FUNCTION_BLOCK ConveyorSC_NC
VAR_INPUT
	bEnable : BOOL;
END_VAR
VAR_OUTPUT
	sensorEntry AT %I* : BOOL := TRUE;
	sensorExit AT %I* : BOOL := TRUE;
	
	trueMode : ConveyorMode;
	requestedMode : ConveyorMode;
	
	position : LREAL;
	velocity : LREAL;
	ready : BOOL;
END_VAR
VAR
	axis : AXIS_REF;
	
	mcReadPosition : MC_ReadActualPosition; //continuous enable FBs
	mcReadVelocity : MC_ReadActualVelocity;
	mcReadError : MC_ReadAxisError;
	mcPower : MC_Power;
	
	mcReset : MC_Reset; //rising edge FBs
	mcMoveAbsolute : MC_MoveAbsolute;
	mcMoveRelative : MC_MoveRelative;
	mcMoveVelocity : MC_MoveVelocity;
	
	mcSetPosition : MC_SetPosition;
	mcStop : MC_Stop;
END_VAR
VAR_STAT CONSTANT
	targetingVelocity : INT := 500;
	continuousVelocity : INT := 500;
END_VAR
(*
this FB represents a standard slat conveyor with no lifter
	compliant with PLCopen motion control

unlike standalone servos,
	conveyors need to coordinate (not slave) their motion with other conveyors
	and be able to set their current position to any value as required by the system
	
moveAbsolute is provided for now but should not be used for position targetting and may be protected/privated later
instead, request/set the operation mode and the motion will follow
*)

IF error THEN
	stop();
	reset();
	
ELSE
	CASE trueMode OF
		ConveyorMode.IDLE:			stop();	
		ConveyorMode.FORWARD:		moveContinuous(direction:= MC_Positive_Direction);
		ConveyorMode.BACKWARD:		moveContinuous(direction:= MC_Negative_Direction);
		ConveyorMode.STOP:			stop();
	END_CASE
	
END_IF

blocks();

mcReset.Execute := FALSE;
mcMoveAbsolute.Execute := FALSE;
mcMoveRelative.Execute := FALSE;
mcMoveVelocity.Execute := FALSE;
mcSetPosition.Execute := FALSE;
mcStop.Execute := FALSE;

blocks();

PROPERTY Active : BOOL
GET
Active := 
	mcMoveAbsolute.Busy OR 
	mcMoveRelative.Busy OR 
	mcMoveVelocity.Busy OR 
	mcSetPosition.Busy OR 
	mcReset.Busy OR 
	mcStop.Busy;
END_GET
END_PROPERTY

METHOD PRIVATE blocks : BOOL
mcReadPosition(
	Axis:= axis, 
	Enable:= TRUE, 
	Valid=> , 
	Busy=> , 
	Error=> , 
	ErrorID=> , 
	Position=> position);
	
mcReadVelocity(
	Axis:= axis, 
	Enable:= TRUE, 
	Valid=> , 
	Busy=> , 
	Error=> , 
	ErrorID=> , 
	ActualVelocity=> velocity);
	
mcReadError(
	Axis:= axis, 
	Enable:= TRUE, 
	Valid=> , 
	Busy=> , 
	Error=> , 
	ErrorID=> , 
	AxisErrorID=> );
	
mcPower(
	Axis:= axis, 
	Enable:= bEnable, 
	Enable_Positive:= TRUE, 
	Enable_Negative:= TRUE, 
	Override:= 100, 
	BufferMode:= , 
	Options:= , 
	Status=> , 
	Busy=> , 
	Active=> , 
	Error=> , 
	ErrorID=> );

mcReset(
	Axis:= axis, 
	Execute:= , 
	Done=> , 
	Busy=> , 
	Error=> , 
	ErrorID=> );

mcMoveAbsolute(
	Axis:= axis, 
	Execute:= , 
	Position:= , 
	Velocity:= targetingVelocity, 
	Acceleration:= , 
	Deceleration:= , 
	Jerk:= , 
	BufferMode:= , 
	Options:= , 
	Done=> , 
	Busy=> , 
	Active=> , 
	CommandAborted=> , 
	Error=> , 
	ErrorID=> );
	
mcMoveRelative(
	Axis:= axis, 
	Execute:= , 
	Distance:= ,
	Velocity:= targetingVelocity, 
	Acceleration:= , 
	Deceleration:= , 
	Jerk:= , 
	BufferMode:= , 
	Options:= , 
	Done=> , 
	Busy=> , 
	Active=> , 
	CommandAborted=> , 
	Error=> , 
	ErrorID=> );
	
mcMoveVelocity( //stopped with stop();
	Axis:= axis, 
	Execute:= , 
	Velocity:= continuousVelocity, 
	Acceleration:= , 
	Deceleration:= , 
	Jerk:= , 
	Direction:= , 
	BufferMode:= , 
	Options:= , 
	InVelocity=> , 
	Busy=> , 
	Active=> , 
	CommandAborted=> , 
	Error=> , 
	ErrorID=> );
	
mcSetPosition(
	Axis:= axis, 
	Execute:= , 
	Position:= , 
	Mode:= , 
	Options:= , 
	Done=> , 
	Busy=> , 
	Error=> , 
	ErrorID=> );
	
mcStop(
	Axis:= axis, 
	Execute:= , 
	Deceleration:= , 
	Jerk:= , 
	Options:= , 
	Done=> , 
	Busy=> , 
	Active=> , 
	CommandAborted=> , 
	Error=> , 
	ErrorID=> );
END_METHOD

PROPERTY CurrentPosition : LREAL
GET
CurrentPosition := position;
END_GET
SET
position := CurrentPosition;
END_SET
END_PROPERTY

PROPERTY Error : BOOL
GET
error := 
	mcMoveAbsolute.Error OR 
	mcMoveRelative.Error OR 
	mcMoveVelocity.Error OR 
	mcSetPosition.Error OR 
	mcReset.Error OR 
	mcStop.Error OR
	mcReadError.AxisErrorID > 0;
END_GET
END_PROPERTY

{attribute 'monitoring' := 'call'}
PROPERTY IsOccupied : BOOL
GET
IsOccupied := sensorExit OR sensorEntry;
END_GET
END_PROPERTY

METHOD moveAbsolute : BOOL
VAR_INPUT
	newTarget : LREAL;
END_VAR
mcMoveAbsolute.Position := newTarget;

IF NOT Active AND NOT error THEN
	mcMoveAbsolute.Execute := TRUE;
END_IF

moveAbsolute := 
	//mcMoveAbsolute.Done;
	CurrentPosition = TargetPosition;
END_METHOD

METHOD moveContinuous : BOOL
VAR_INPUT
	direction : MC_Direction;
END_VAR
mcMoveVelocity.Direction := direction;

IF NOT Active AND NOT error THEN
	mcMoveVelocity.Execute := TRUE;
	moveContinuous := TRUE;
END_IF
END_METHOD

METHOD reset : BOOL
VAR_INPUT
END_VAR
mcReset.Execute := TRUE;

reset := mcReset.Done;
END_METHOD

METHOD setMode : BOOL
VAR_INPUT
	mode : ConveyorMode;
END_VAR
trueMode := mode;
END_METHOD

METHOD setRequest : BOOL
VAR_INPUT
	newRequest : ConveyorMode;
END_VAR
requestedMode := newRequest;
END_METHOD

METHOD stop : BOOL
VAR_INPUT
END_VAR
mcStop.Execute := TRUE;

mcMoveAbsolute.Execute := FALSE;
mcMoveRelative.Execute := FALSE;
mcMoveVelocity.Execute := FALSE;
END_METHOD

PROPERTY TargetPosition : LREAL
GET
END_GET
SET
moveAbsolute(newTarget := TargetPosition);
END_SET
END_PROPERTY

END_FUNCTION_BLOCK

(* stored: Version 1.1.0.1, ProductVersion 3.1.4024.11
   POU ConveyorSC_NC: Id {1a3c206e-0069-4a63-babe-f3447b402daa}, SpecialFunc None
   Folder OpMode: Id {7126b177-f7bc-483e-a256-95db5f12c9e4}
   Folder Private: Id {27aadce1-d903-452f-adb2-54f83ddb3a5f}
   Folder Properties: Id {fc9cf1c4-a3bd-45bb-98c1-7e5f7668ac56}
   Property Active: Id {8577ae16-3f9d-4ebf-87f7-665ddde652c7}
   Get Get: Id {fda9c8e0-be6a-4c77-ab1c-5aee09adb92c}
   Method blocks: Id {5e2d39b4-dd14-4752-a684-95c0c1657fc2}
   Property CurrentPosition: Id {91176e7f-8c37-4654-ae4a-37c923738f16}
   Get Get: Id {daa93656-cb6e-4912-a464-1654f86ffd26}
   Set Set: Id {c9022b20-e9cd-4a9c-99e3-78163e746db2}
   Property Error: Id {17949c08-c0bf-41ef-bbc6-5c7512a312ee}
   Get Get: Id {05305283-5e7a-42ce-9f39-02b3a802344d}
   Property IsOccupied: Id {fa852f38-dc7b-45c2-a409-f05c12c19ba6}
   Get Get: Id {1a019571-aaa0-4752-990b-625c112713fd}
   Method moveAbsolute: Id {890fa2cb-8f94-4e6f-8a1d-a12b54a341ab}
   Method moveContinuous: Id {fcb4ecba-00d9-4b29-9ddc-24c3b2555d93}
   Method reset: Id {c7e6f6a2-38c5-4a94-8683-e5362479dd88}
   Method setMode: Id {44be4b30-7778-4d9e-bcd2-ac7c57f30f08}
   Method setRequest: Id {a7a6efa5-83c8-4394-aa6b-cbbdb4d865d8}
   Method stop: Id {2153e19f-9e1a-430b-9392-9f8b157e93fb}
   Property TargetPosition: Id {96dde37d-ab48-4cb5-8241-1a2ed5f503b8}
   Get Get: Id {e8b2fd3d-b8b4-4412-a8d1-07730f90936c}
   Set Set: Id {98ece328-8848-405c-a0c3-d9ad9e7e12c8} *)
